# EPICS substitutions: iocBoot/iocMksu/mksu.substitutions
file ../../db/mksu.template
{
pattern
{AREA, LOCATION, PORT, CHANNEL, TIMEOUT, SCAN}
#{1, 1, Mksu, 0, 1, "I/O Intr"}
#{IN20, 3130, Mksu, 0, 1, "1 second"}
{1, 1, Mksu, 0, 1, ".1 second"}
}
